FUNCTION_BLOCK "Semantic_VariantInStatic"
{ S7_Optimized_Access := 'TRUE' }
VERSION : 0.1

VAR
    badVariant : Variant;
    // EXPECT: error[type.illegal-section] SEM-SECTION-001
END_VAR

BEGIN
END_FUNCTION_BLOCK
